{attribute addProperty BoxType "EL6201-0000-0017"}
{attribute addProperty Id "Slave_2A_DI0BIT10.1259Slave_2A_DI1BIT10.12510Slave_2A_DI2BIT10.12511Slave_2A_DI3BIT10.12512Slave_2B_DI0BIT10.12513Slave_2B_DI1BIT10.12514Slave_2B_DI2BIT10.12515Slave_2B_DI3BIT10.12516"}
{attribute addProperty CRC "850247186"}
{attribute addProperty SizeInBites "8"}
{attribute addProperty SizeInBytes "1"}
TYPE Slave_2_Inputs_32ADBE12 :
STRUCT
	{attribute addProperty Name "Slave_2A_DI0"}
	Slave_2A_DI0 : BIT;
	{attribute addProperty Name "Slave_2A_DI1"}
	Slave_2A_DI1 : BIT;
	{attribute addProperty Name "Slave_2A_DI2"}
	Slave_2A_DI2 : BIT;
	{attribute addProperty Name "Slave_2A_DI3"}
	Slave_2A_DI3 : BIT;
	{attribute addProperty Name "Slave_2B_DI0"}
	Slave_2B_DI0 : BIT;
	{attribute addProperty Name "Slave_2B_DI1"}
	Slave_2B_DI1 : BIT;
	{attribute addProperty Name "Slave_2B_DI2"}
	Slave_2B_DI2 : BIT;
	{attribute addProperty Name "Slave_2B_DI3"}
	Slave_2B_DI3 : BIT;
END_STRUCT
END_TYPE

(* stored: Version 1.2.0.0, ProductVersion 3.1.4024.9
   DUT Slave_2_Inputs_32ADBE12: Id {b1fa00dc-1e39-4147-a4b9-cec9fd61b6e2} *)
